// Mitsubishi GX Works2 project: Prática 03 - MOTOR   PLC: FX3U/FX3UC
// Configuração Modbus RTU

PROGRAM MAIN
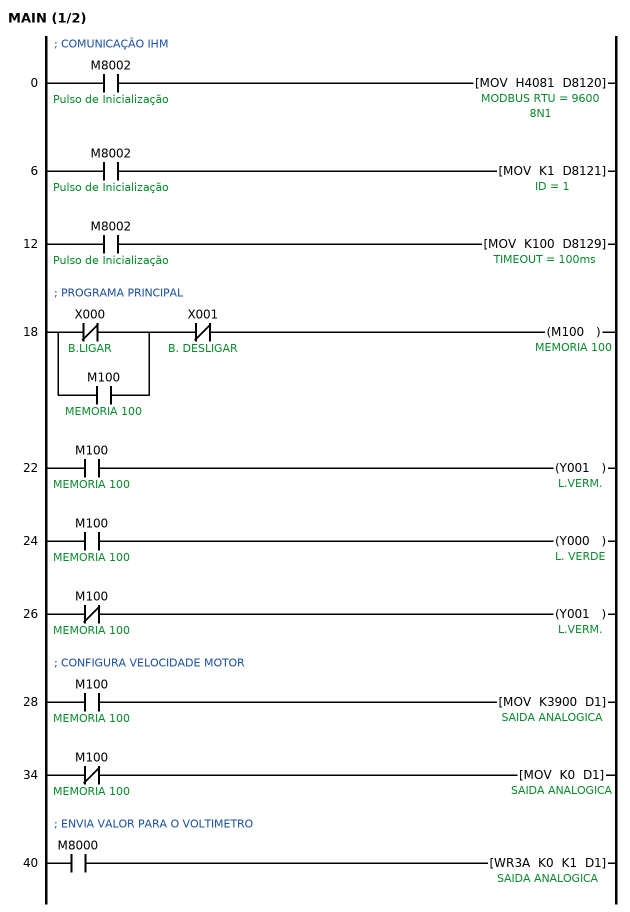
; COMUNICAÇÃO IHM
0     LD      M8002  ; Pulso de Inicialização
      MOV     H4081 D8120  ; MODBUS RTU = 9600 8N1
6     LD      M8002  ; Pulso de Inicialização
      MOV     K1 D8121  ; ID = 1
12    LD      M8002  ; Pulso de Inicialização
      MOV     K100 D8129  ; TIMEOUT = 100ms
; PROGRAMA PRINCIPAL
18    LDI     X000  ; B.LIGAR
      OR      M100  ; MEMORIA 100
      ANI     X001  ; B. DESLIGAR
      OUT     M100  ; MEMORIA 100
22    LD      M100  ; MEMORIA 100
      OUT     Y001  ; L.VERM.
24    LD      M100  ; MEMORIA 100
      OUT     Y000  ; L. VERDE
26    LDI     M100  ; MEMORIA 100
      OUT     Y001  ; L.VERM.
; CONFIGURA VELOCIDADE MOTOR
28    LD      M100  ; MEMORIA 100
      MOV     K3900 D1  ; SAIDA ANALOGICA
34    LDI     M100  ; MEMORIA 100
      MOV     K0 D1
; ENVIA VALOR PARA O VOLTIMETRO
40    LD      M8000
      WR3A    K0 K1 D1
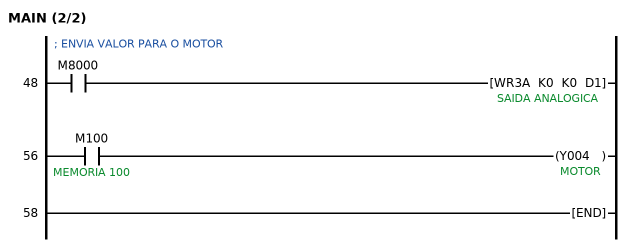
; ENVIA VALOR PARA O MOTOR
48    LD      M8000
      WR3A    K0 K0 D1
56    LD      M100  ; MEMORIA 100
      OUT     Y004  ; MOTOR
58    END
END_PROGRAM

// device comments not shown above
Y002  ; RELE 2
Y005  ; SENTIDO
M0  ; VARIAVEL DE MEMORIA 0
M1  ; VARIAVEL DE MEMORIA 1
M2  ; VARIAVEL DE MEMORIA 2
D0  ; REGISTRO 0
D2  ; ENCHE O TANQUE
D3  ; ESVAZIA O TANQUE
